Staubli VAL3: testApp.pjx

Parameters version=s7.9.1 stackSize=5000 millimeterUnit=true
Program file=start.pgx
Program file=stop.pgx
Data file=testApp.dtx
